(*
Grundfos CM pump that can be switch on/off
*)

FUNCTION_BLOCK Pump_GrundfosCM EXTENDS FB_Actor2Point
VAR
	//I/O Links
	bSetStatusOn_OUT 	AT %Q* : BOOL := FALSE;
END_VAR

METHOD SetState_BO : BOOL
VAR_INPUT
END_VAR
//control state
controlState.bStatusOn := bSetStatusOn; //pump does not have a status module, so control state gets internal bSetStatusOn variable

//output
bSetStatusOn_OUT := bSetStatusOn;
END_METHOD

END_FUNCTION_BLOCK

(* stored: Version 1.1.0.1, ProductVersion 3.1.4024.9
   POU Pump_GrundfosCM: Id {5b6d9bd2-ce18-456b-8ae2-afbacf79793a}, SpecialFunc None
   Method SetState_BO: Id {36b0dedc-9e39-443a-8eb0-332e87306b63} *)
